{attribute 'qualified_only'}
{attribute 'strict'}
{attribute 'to_string'}
TYPE E_MOVER_SELECTOR :
(
	SELECT_MOVER_INDEX,
  SELECT_MOVER_AXIS_ID
);
END_TYPE

(* stored: Version 1.1.0.1, ProductVersion 3.1.4026.13
   DUT E_MOVER_SELECTOR: Id {488fac83-78dd-4907-b8e7-a4a8007f9fea} *)
